FUNCTION_BLOCK T_Stream IMPLEMENTS I_Stream, I_StreamWriter, I_StreamReader
VAR

    MemoryManager : FB_DynMem_Manager;
    Buffer        : FB_DynMem_Buffer(ipMemMan := MemoryManager);
    pBuffer       : POINTER TO BYTE;

    _StreamLength : UDINT := 4;
    _Position     : UDINT;
END_VAR

METHOD PRIVATE _Resize
VAR_INPUT
    StreamLength : UDINT;
END_VAR
Buffer.Resize(nSize     := StreamLength,
              bPreserve := TRUE,
              bReset    := FALSE);

_StreamLength := StreamLength;
pBuffer       := Buffer.pBuffer;
END_METHOD

METHOD PRIVATE _ResizeIfNecessary
VAR_INPUT
    SpaceRequired : UDINT;
END_VAR
IF _Position + SpaceRequired > _StreamLength THEN
    _Resize(StreamLength := _StreamLength * 2);
END_IF
END_METHOD

METHOD Add_BLOB : I_StreamWriter
VAR_INPUT
    Value : ANY;
END_VAR
VAR
    pValue : POINTER TO BYTE;
END_VAR
_ResizeIfNecessary(SpaceRequired := DINT_TO_UDINT(Value.diSize));

MEMCPY(destAddr := pBuffer + _Position,
       srcAddr  := Value.pValue,
       n        := DINT_TO_UDINT(Value.diSize));

_Position := _Position + DINT_TO_UDINT(Value.diSize);

Add_BLOB := THIS^;
END_METHOD

METHOD Add_BOOL : I_StreamWriter
VAR_INPUT
    Value : BOOL;
END_VAR
VAR
    pValue : POINTER TO BOOL;
END_VAR
_ResizeIfNecessary(SpaceRequired := SIZEOF(Value));

pValue    := pBuffer + _Position;
pValue^   := Value;
_Position := _Position + SIZEOF(Value);

Add_BOOL := THIS^;
END_METHOD

METHOD Add_BYTE : I_StreamWriter
VAR_INPUT
    Value : BYTE;
END_VAR
VAR
    pValue : POINTER TO BYTE;
END_VAR
_ResizeIfNecessary(SpaceRequired := SIZEOF(Value));

pValue    := pBuffer + _Position;
pValue^   := Value;
_Position := _Position + SIZEOF(Value);

Add_BYTE := THIS^;
END_METHOD

METHOD Add_DINT : I_StreamWriter
VAR_INPUT
    Value : DINT;
END_VAR
VAR
    pValue : POINTER TO DINT;
END_VAR
_ResizeIfNecessary(SpaceRequired := SIZEOF(Value));

pValue    := pBuffer + _Position;
pValue^   := Value;
_Position := _Position + SIZEOF(Value);

Add_DINT := THIS^;
END_METHOD

METHOD Add_INT : I_StreamWriter
VAR_INPUT
    Value : INT;
END_VAR
VAR
    pValue : POINTER TO INT;
END_VAR
_ResizeIfNecessary(SpaceRequired := SIZEOF(Value));

pValue    := pBuffer + _Position;
pValue^   := Value;
_Position := _Position + SIZEOF(Value);

Add_INT := THIS^;
END_METHOD

METHOD Add_LINT : I_StreamWriter
VAR_INPUT
    Value : LINT;
END_VAR
VAR
    pValue : POINTER TO LINT;
END_VAR
_ResizeIfNecessary(SpaceRequired := SIZEOF(Value));

pValue    := pBuffer + _Position;
pValue^   := Value;
_Position := _Position + SIZEOF(Value);

Add_LINT := THIS^;
END_METHOD

METHOD Add_LREAL : I_StreamWriter
VAR_INPUT
    Value : LREAL;
END_VAR
VAR
    pValue : POINTER TO LREAL;
END_VAR
_ResizeIfNecessary(SpaceRequired := SIZEOF(Value));

pValue    := pBuffer + _Position;
pValue^   := Value;
_Position := _Position + SIZEOF(Value);

Add_LREAL := THIS^;
END_METHOD

METHOD Add_PVOID : I_StreamWriter
VAR_INPUT
    Value : PVOID;
END_VAR
VAR
    pValue : POINTER TO PVOID;
END_VAR
_ResizeIfNecessary(SpaceRequired := SIZEOF(Value));

pValue    := pBuffer + _Position;
pValue^   := Value;
_Position := _Position + SIZEOF(Value);

Add_PVOID := THIS^;
END_METHOD

METHOD Add_REAL : I_StreamWriter
VAR_INPUT
    Value : REAL;
END_VAR
VAR
    pValue : POINTER TO REAL;
END_VAR
_ResizeIfNecessary(SpaceRequired := SIZEOF(Value));

pValue    := pBuffer + _Position;
pValue^   := Value;
_Position := _Position + SIZEOF(Value);

Add_REAL := THIS^;
END_METHOD

METHOD Add_STRING : I_StreamWriter // adds any string length as we only store the chars + null byte
VAR_INPUT
    Value : STRING(255);
END_VAR
VAR
    StringSize : UDINT; // number of characters plus the null termination byte
END_VAR
StringSize := INT_TO_UDINT(LEN(Value) + 1);

_ResizeIfNecessary(SpaceRequired := StringSize); // only storing the characters and the null termination byte

MEMCPY(destAddr := pBuffer + _Position,
       srcAddr  := ADR(Value),
       n        := StringSize);

_Position := _Position + StringSize;

Add_STRING := THIS^;
END_METHOD

METHOD Add_UDINT : I_StreamWriter
VAR_INPUT
    Value : UDINT;
END_VAR
VAR
    pValue : POINTER TO UDINT;
END_VAR
_ResizeIfNecessary(SpaceRequired := SIZEOF(Value));

pValue    := pBuffer + _Position;
pValue^   := Value;
_Position := _Position + SIZEOF(Value);

Add_UDINT := THIS^;
END_METHOD

METHOD Add_UINT : I_StreamWriter
VAR_INPUT
    Value : UINT;
END_VAR
VAR
    pValue : POINTER TO UINT;
END_VAR
_ResizeIfNecessary(SpaceRequired := SIZEOF(Value));

pValue    := pBuffer + _Position;
pValue^   := Value;
_Position := _Position + SIZEOF(Value);

Add_UINT := THIS^;
END_METHOD

METHOD Add_ULINT : I_StreamWriter
VAR_INPUT
    Value : ULINT;
END_VAR
VAR
    pValue : POINTER TO ULINT;
END_VAR
_ResizeIfNecessary(SpaceRequired := SIZEOF(Value));

pValue    := pBuffer + _Position;
pValue^   := Value;
_Position := _Position + SIZEOF(Value);

Add_ULINT := THIS^;
END_METHOD

PROPERTY BufferAddress : PVOID
GET
BufferAddress := pBuffer;
END_GET
END_PROPERTY

METHOD Clear : I_StreamWriter
Buffer.Clear();
_Position := 0;
pBuffer   := Buffer.pBuffer;
Clear     := THIS^;
END_METHOD

METHOD CopyFrom
VAR_INPUT
    StreamToCopyFrom : I_Stream;
END_VAR
IF StreamToCopyFrom <> 0 THEN
    IF StreamToCopyFrom.StreamLength > THIS^.StreamLength THEN
        _Resize(StreamToCopyFrom.StreamLength);
    END_IF

    MEMCPY(destAddr := Buffer.pBuffer,
           srcAddr  := StreamToCopyFrom.BufferAddress,
           n        := StreamToCopyFrom.StreamLength);

    THIS^._StreamLength := StreamToCopyFrom.StreamLength;
    THIS^._Position     := 0;
END_IF
END_METHOD

METHOD FB_exit : BOOL
VAR_INPUT
	bInCopyCode : BOOL; // if TRUE, the exit method is called for exiting an instance that is copied afterwards (online change).
END_VAR
IF NOT bInCopyCode THEN
    Buffer.DeleteBuffer();
END_IF
END_METHOD

METHOD FB_init : BOOL
VAR_INPUT
    bInitRetains : BOOL; // if TRUE, the retain variables are initialized (warm start / cold start)
    bInCopyCode  : BOOL; // if TRUE, the instance afterwards gets moved into the copy code (online change)
    StreamLength : UDINT;
END_VAR
IF NOT bInCopyCode THEN
    Init(StreamLength);
END_IF
END_METHOD

METHOD GetNextArgTypeId : E_ArgTypeId;
VAR
    pValue : POINTER TO INT;
    Result : INT;
END_VAR
IF _Position + SIZEOF(Result) <= _StreamLength THEN
    pValue           := pBuffer + _Position;
    Result           := pValue^;
    _Position        := _Position + SIZEOF(Result);
    GetNextArgTypeId := Result;
END_IF
END_METHOD

METHOD Init
VAR_INPUT
    StreamLength : UDINT;
END_VAR
IF Buffer.bAvailable THEN
    Buffer.DeleteBuffer();
END_IF

_StreamLength := StreamLength;
Buffer.CreateBuffer(nSize  := _StreamLength,
                    bReset := TRUE);

_Position := 0;
pBuffer   := Buffer.pBuffer;
END_METHOD

PROPERTY Position : UDINT
GET
Position := _Position;
END_GET
END_PROPERTY

METHOD Read_BLOB
VAR_INPUT
    Value : ANY;
END_VAR
VAR
    pValue : POINTER TO BYTE;
END_VAR
IF _Position + DINT_TO_UDINT(Value.diSize) <= _StreamLength THEN
    MEMCPY(destAddr := Value.pValue,
           srcAddr  := pBuffer + _Position,
           n        := DINT_TO_UDINT(Value.diSize));

    _Position := _Position + DINT_TO_UDINT(Value.diSize);
END_IF
END_METHOD

METHOD Read_BOOL : BOOL;
VAR
    pValue : POINTER TO BOOL;
    Result : BOOL;
END_VAR
IF _Position + SIZEOF(Result) <= _StreamLength THEN
	pValue    := pBuffer + _Position;
	Result    := pValue^;
	_Position := _Position + SIZEOF(Result);
	Read_BOOL := Result;
END_IF
END_METHOD

METHOD Read_BYTE : BYTE;
VAR
    pValue : POINTER TO BYTE;
    Result : BYTE;
END_VAR
IF _Position + SIZEOF(Result) <= _StreamLength THEN
	pValue    := pBuffer + _Position;
	Result    := pValue^;
	_Position := _Position + SIZEOF(Result);
	Read_BYTE := Result;
END_IF
END_METHOD

METHOD Read_DINT : DINT;
VAR
    pValue : POINTER TO DINT;
    Result : DINT;
END_VAR
IF _Position + SIZEOF(Result) <= _StreamLength THEN
	pValue    := pBuffer + _Position;
	Result    := pValue^;
	_Position := _Position + SIZEOF(Result);
	Read_DINT := Result;
END_IF
END_METHOD

METHOD Read_INT : INT;
VAR
    pValue : POINTER TO INT;
    Result : INT;
END_VAR
IF _Position + SIZEOF(Result) <= _StreamLength THEN
	pValue    := pBuffer + _Position;
	Result    := pValue^;
	_Position := _Position + SIZEOF(Result);
	Read_INT  := Result;
END_IF
END_METHOD

METHOD Read_LINT : LINT;
VAR
    pValue : POINTER TO LINT;
    Result : LINT;
END_VAR
IF _Position + SIZEOF(Result) <= _StreamLength THEN
	pValue    := pBuffer + _Position;
	Result    := pValue^;
	_Position := _Position + SIZEOF(Result);
	Read_LINT := Result;
END_IF
END_METHOD

METHOD Read_LREAL : LREAL;
VAR
    pValue : POINTER TO LREAL;
    Result : LREAL;
END_VAR
IF _Position + SIZEOF(Result) <= _StreamLength THEN
	pValue     := pBuffer + _Position;
	Result     := pValue^;
	_Position  := _Position + SIZEOF(Result);
	Read_LREAL := Result;
END_IF
END_METHOD

METHOD Read_PVOID : PVOID;
VAR
    pValue : POINTER TO PVOID;
    Result : PVOID;
END_VAR
IF _Position + SIZEOF(Result) <= _StreamLength THEN
	pValue     := pBuffer + _Position;
	Result     := pValue^;
	_Position  := _Position + SIZEOF(Result);
	Read_PVOID := Result;
END_IF
END_METHOD

METHOD Read_REAL : REAL;
VAR
    pValue : POINTER TO REAL;
    Result : REAL;
END_VAR
IF _Position + SIZEOF(Result) <= _StreamLength THEN
	pValue    := pBuffer + _Position;
	Result    := pValue^;
	_Position := _Position + SIZEOF(Result);
	Read_REAL := Result;
END_IF
END_METHOD

METHOD Read_STRING : STRING(255);
VAR
    pValue : POINTER TO STRING(255);
    StringSize : UDINT; // number of characters plus the null termination byte
END_VAR
pValue     := pBuffer + _Position;
StringSize := INT_TO_UDINT(LEN(pValue^) + 1);
IF _Position + StringSize <= _StreamLength THEN // end of string is in the buffer, so proceed...
	_Position   := _Position + StringSize;
	Read_STRING := pValue^;
END_IF
END_METHOD

METHOD Read_UDINT : UDINT;
VAR
    pValue : POINTER TO UDINT;
    Result : UDINT;
END_VAR
IF _Position + SIZEOF(Result) <= _StreamLength THEN
	pValue     := pBuffer + _Position;
	Result     := pValue^;
	_Position  := _Position + SIZEOF(Result);
	Read_UDINT := Result;
END_IF
END_METHOD

METHOD Read_UINT : UINT;
VAR
    pValue : POINTER TO UINT;
    Result : UINT;
END_VAR
IF _Position + SIZEOF(Result) <= _StreamLength THEN
	pValue    := pBuffer + _Position;
	Result    := pValue^;
	_Position := _Position + SIZEOF(Result);
	Read_UINT := Result;
END_IF
END_METHOD

METHOD Read_ULINT : ULINT;
VAR
    pValue : POINTER TO ULINT;
    Result : ULINT;
END_VAR
IF _Position + SIZEOF(Result) <= _StreamLength THEN
	pValue     := pBuffer + _Position;
	Result     := pValue^;
	_Position  := _Position + SIZEOF(Result);
	Read_ULINT := Result;
END_IF
END_METHOD

METHOD Seek : I_StreamWriter
VAR_INPUT
    Position : UDINT;
END_VAR
IF Position <= _StreamLength THEN
    THIS^._Position := Position;
END_IF
Seek := THIS^;
END_METHOD

METHOD SetNextArgTypeId : I_StreamWriter
VAR_INPUT
    Value : E_ArgTypeId;
END_VAR
VAR
    pValue : POINTER TO INT;
END_VAR
_ResizeIfNecessary(SpaceRequired := SIZEOF(Value));

pValue    := pBuffer + _Position;
pValue^   := Value;
_Position := _Position + SIZEOF(Value);

SetNextArgTypeId := THIS^;
END_METHOD

PROPERTY StreamLength : UDINT
GET
StreamLength := _StreamLength;
END_GET
END_PROPERTY

END_FUNCTION_BLOCK

(* stored: Version 1.1.0.1, ProductVersion 3.1.4024.6
   POU T_Stream: Id {7de9e7b4-a803-0786-2483-a2ef3055cb50}, SpecialFunc None
   Folder Methods: Id {3607c258-fd4e-0eca-0c2c-f6847ad6a5df}
   Folder Properties: Id {0109ea30-a082-4efa-bae3-f69dc56d1ba2}
   Method _Resize: Id {6eedcc64-a81c-456d-b6ba-eafb61d80242}
   Method _ResizeIfNecessary: Id {4c85beec-fafd-0332-0264-65f3f9273dc7}
   Method Add_BLOB: Id {eb34da3f-d27f-4e89-869e-adb85eec5235}
   Method Add_BOOL: Id {7beb3c3e-8d84-0c46-1458-1b7b92b63e30}
   Method Add_BYTE: Id {030e1fb0-78e9-06d1-01fb-084ed99a7c86}
   Method Add_DINT: Id {31239b38-361b-0d3f-0af3-2f3ef2e9e59b}
   Method Add_INT: Id {f9865655-2cea-04b1-0a9e-c5b2fbf2b477}
   Method Add_LINT: Id {1820a32d-1cd7-0625-2cfd-f88d8a948838}
   Method Add_LREAL: Id {2d9ba739-a603-01e0-21a0-2f35e9c49f5a}
   Method Add_PVOID: Id {371876cd-4ebf-0d9d-1f20-40f781dfe335}
   Method Add_REAL: Id {473baad3-6290-0f2e-0f58-01351f75f993}
   Method Add_STRING: Id {21b62581-7a37-0bd9-1176-a322997395f8}
   Method Add_UDINT: Id {2f4586aa-cb30-039c-24e6-bbfc08c0c422}
   Method Add_UINT: Id {7b471ebb-85a2-0c54-0eda-e85c8d920fc4}
   Method Add_ULINT: Id {3b924970-9e4f-0249-16d4-29cce8f96575}
   Property BufferAddress: Id {5f457907-a510-4dbe-8c24-29101ff67677}
   Get Get: Id {1d8dfcf7-ea78-4390-8987-d61b96c8ce39}
   Method Clear: Id {aa527d30-0b4c-08d4-1da8-932172a4f081}
   Method CopyFrom: Id {628a2f83-9063-4b54-963c-41529f121199}
   Method FB_exit: Id {6fe0ad89-3a2a-067e-3d39-721acf587bbb}
   Method FB_init: Id {64f819ea-8af0-05ad-3ef0-540d0e10a939}
   Method GetNextArgTypeId: Id {37e01e90-358e-43fb-9f34-5890d2d4cee9}
   Method Init: Id {2b40521b-bf8d-0ff7-031c-928f3bdfedb6}
   Property Position: Id {66f9b2cc-0047-4e43-b894-a659d2355adb}
   Get Get: Id {e1f72485-462d-4053-a202-09eef1285a86}
   Method Read_BLOB: Id {6c7c1fdf-c083-4215-bc18-a8edadcb5fa1}
   Method Read_BOOL: Id {af54e0cd-16dd-0373-2061-97f060da1982}
   Method Read_BYTE: Id {2f79e8aa-a1ce-0388-3637-aca716c1825f}
   Method Read_DINT: Id {52b2e8be-af73-0b66-3ede-3e6c6875df1d}
   Method Read_INT: Id {88f59eaf-d475-0936-0514-fd747bd37737}
   Method Read_LINT: Id {9b94dfea-162d-0221-05c6-083e6fc3a489}
   Method Read_LREAL: Id {8b3953c5-1588-0a54-23ab-12e037540a96}
   Method Read_PVOID: Id {cbb33155-c6b1-0f12-39f0-968b46d8481d}
   Method Read_REAL: Id {68d4b51d-5637-03b3-2b8a-130f04bf24e9}
   Method Read_STRING: Id {4fbbee87-6322-0666-117c-f80beac8fb2a}
   Method Read_UDINT: Id {bc064b6d-c61a-0649-34a8-7347e22bc625}
   Method Read_UINT: Id {307605e7-bec9-0e51-20c3-ea75a90ec7f4}
   Method Read_ULINT: Id {cf5324b0-9555-098c-1d59-f105b6163144}
   Method Seek: Id {00a3579c-6e96-0aa2-0dc9-f99eba3a69fc}
   Method SetNextArgTypeId: Id {79a85dde-c616-420f-8dca-96cad7e7b06f}
   Property StreamLength: Id {392a552a-86e8-4535-bed7-6e59ef8ae550}
   Get Get: Id {831bcec9-b5f7-4dcc-ad53-7002fdda3d3a} *)
